// TIA Portal project "3 Animation final project" (V13)

(* hardware
DEVICE "S7-1200 station_1"  S7-1200 Station
   slot 0: "Rack_0"  Rack  V1.0
   slot 1: "PLC_1"  CPU 1212C AC/DC/Rly  6ES7 212-1BE40-0XB0  V4.1
DEVICE "HMI_1"  KTP400 Basic PN
   slot 0: "HMI"  HMI  6AV2 123-2DB03-0AX0  13.0.1.0
   slot 1: "HMI_RT_1"  KTP400 Basic PN  6AV2 123-2DB03-0AX0  13.0.1.0
   slot 5: "HMI_1.IE_CP_1"  PROFINET Interface
      slot 1: "PROFINET Interface_1"  PROFINET Interface
         slot 1: "Port_1"  Port
*)

// ===== PLC "PLC_1"  CPU 1212C AC/DC/Rly =====

VAR_GLOBAL   // PLC tag table "Default tag table"
   "Tag_1" AT %MD5 : DWord;
   "Tag_2" AT %MD0 : DWord;
   "Tag_4" AT %MW5 : Word;
   "Tag_3" AT %MW10 : Int;
   "Move box right" AT %M100.0 : Bool;
   "Motor up" AT %Q0.0 : Bool;
   "Move box left" AT %M100.1 : Bool;
   "Motor anti clockwise" AT %Q0.1 : Bool;
   "Tag_9" AT %MD5 : Time;
   "Tag_10" AT %MD12 : Real;
   "Tag_11" AT %MW15 : Int;
   "Capacitive Analog" AT %ID30 : DWord;
   "Tag_13" AT %MD22 : Real;
   "Capacitive Int" AT %MW50 : Word;
   "Motor clockwise" AT %Q0.2 : Bool;
   "Tank Level" AT %ID34 : DWord;
   "Tag_17" AT %MD25 : Real;
   "Tank Level scaled" AT %MD26 : Real;
   "Fill Valve" AT %QD30 : Real;
   "Drain Valve" AT %QD34 : Real;
   "Stop Filling Valve" AT %M200.0 : Bool;
   "Stop Draining Valve" AT %M200.1 : Bool;
   "Animation bit for filling" AT %M40.0 : Bool;
   "Clock_Byte" AT %MB300 : Byte;
   "Clock_10Hz" AT %M300.0 : Bool;
   "Clock_5Hz" AT %M300.1 : Bool;
   "Clock_2.5Hz" AT %M300.2 : Bool;
   "Clock_2Hz" AT %M300.3 : Bool;
   "Clock_1.25Hz" AT %M300.4 : Bool;
   "Clock_1Hz" AT %M300.5 : Bool;
   "Clock_0.625Hz" AT %M300.6 : Bool;
   "Clock_0.5Hz" AT %M300.7 : Bool;
   "Tag_21" AT %MB60 : Byte;
   "roller" AT %MD60 : Real;
   "roller_2" AT %MD70 : Real;
   "Tag_22" AT %MD65 : Real;
   "Tag_23" AT %MW60 : Int;
   "Tag_24" AT %MW65 : Int;
   "Down" AT %M90.0 : Bool;
   "Up" AT %M90.1 : Bool;
   "Door Animation Bit" AT %MW75 : Int;
   "Tag_26" AT %MW78 : Int;
   "Tag_27" AT %MW80 : Int;
   "Down(1)" AT %M90.2 : Bool;
   "Motor down" AT %Q0.3 : Bool;
   "Door Motor bit" AT %M101.0 : Bool;
END_VAR

// folder: System blocks/Program resources

DATA_BLOCK "IEC_Timer_0_DB"   // DB1
{ S7_Optimized_Access := 'FALSE' }
AUTHOR : Simatic
FAMILY : IEC
NAME : IEC_TMR
VERSION : 1.0
// stored: InstanceOfName ?
"?"
BEGIN
END_DATA_BLOCK

DATA_BLOCK "IEC_Timer_0_DB_1"   // DB2
{ S7_Optimized_Access := 'FALSE' }
AUTHOR : Simatic
FAMILY : IEC
NAME : IEC_TMR
VERSION : 1.0
// stored: InstanceOfName ?
"?"
BEGIN
END_DATA_BLOCK

DATA_BLOCK "IEC_Timer_0_DB_2"   // DB3
{ S7_Optimized_Access := 'FALSE' }
AUTHOR : Simatic
FAMILY : IEC
NAME : IEC_TMR
VERSION : 1.0
// stored: InstanceOfName ?
"?"
BEGIN
END_DATA_BLOCK

// folder: (top level)

FUNCTION "MHJ-PLC-Lab-Function-S71200" : Void   // FC1, SCL
{ S7_Optimized_Access := 'FALSE' }
VERSION : 0.1
BEGIN

   #Value := PEEK(area := 16#82,
                  dbNumber := 0,
                  byteOffset := 511);
   #Value := #Value + 1;

   POKE(area := 16#82,
        dbNumber := 0,
        byteOffset := 511,
        value := #Value);

   POKE(area := 16#81,
        dbNumber := 0,
        byteOffset := 1016,
        value := #Value_01_DW);
   POKE(area := 16#81,
        dbNumber := 0,
        byteOffset := 1020,
        value := #Value_02_DW);

   POKE(area := 16#81,
        dbNumber := 0,
        byteOffset := 511,
        value := B#16#00);

   FOR #forVal := 0 TO 120 DO
       FOR #forVal_2 := 0 TO 10 DO
           #rdTimeReturn := RD_SYS_T(#outputTime);
           #rdTimeReturn := WR_SYS_T(#outputTime);
           #rdTimeReturn := RD_SYS_T(#outputTime);
           #rdTimeReturn := WR_SYS_T(#outputTime);
       END_FOR;
       #SyncVal := PEEK(area := 16#81,
                        dbNumber := 0,
                        byteOffset := 511);
       IF #SyncVal = #CompVal THEN
           GOTO M_1;
       END_IF;
   END_FOR;
   RETURN;

   M_1:
   POKE(area := 16#81,
        dbNumber := 0,
        byteOffset := 511,
        value := B#16#0);
END_FUNCTION

ORGANIZATION_BLOCK "Main"   // OB1, LAD, ProgramCycle
TITLE = "Main Program Sweep (Cycle)"
{ S7_Optimized_Access := 'FALSE' }
VERSION : 0.1
   VAR_TEMP   // added for the SCL form of the ladder/FBD networks
      _w1 : Bool;
   END_VAR
BEGIN

REGION Network 1: Box Logic
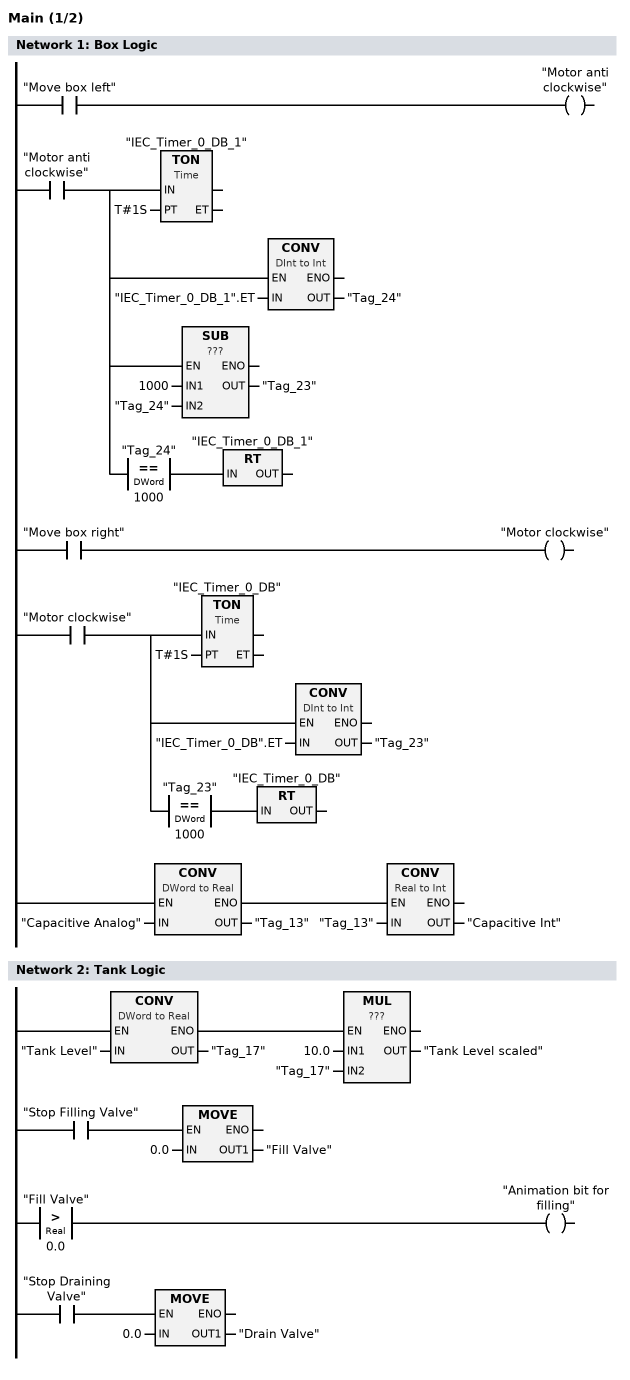
   // ENO of a box is taken as its EN; it also drops when the box reports an error
   "Motor anti clockwise" := "Move box left";
   "IEC_Timer_0_DB_1".TON(IN := "Motor anti clockwise", PT := T#1S);
   IF "Motor anti clockwise" THEN
       "Tag_24" := DINT_TO_INT("IEC_Timer_0_DB_1".ET);
       "Tag_23" := 1000 - "Tag_24";
   END_IF;
   IF "Motor anti clockwise" AND ("Tag_24" = 1000) THEN RESET_TIMER("IEC_Timer_0_DB_1"); END_IF;
   "Motor clockwise" := "Move box right";
   "IEC_Timer_0_DB".TON(IN := "Motor clockwise", PT := T#1S);
   IF "Motor clockwise" THEN "Tag_23" := DINT_TO_INT("IEC_Timer_0_DB".ET); END_IF;
   IF "Motor clockwise" AND ("Tag_23" = 1000) THEN RESET_TIMER("IEC_Timer_0_DB"); END_IF;
   "Tag_13" := DWORD_TO_REAL("Capacitive Analog");
   "Capacitive Int" := REAL_TO_INT("Tag_13");
END_REGION

REGION Network 2: Tank Logic
   RUNG wire#powerrail
      { S7_Templates := "[SrcType := DWord, DestType := Real]"; S7_GenerateENO := "TRUE" } Convert(in := "Tank Level", out => "Tag_17")
      { S7_Templates := "SrcType := ???"; S7_GenerateENO := "TRUE" } Mul(in1 := 10.0, in2 := "Tag_17", out => "Tank Level scaled")
   END_RUNG
   RUNG wire#powerrail
      Contact( "Stop Filling Valve" )
      { S7_GenerateENO := "TRUE" } Move(in := 0.0, out1 => "Fill Valve")
   END_RUNG
   RUNG wire#powerrail
      { S7_Templates := "SrcType := Real" } GT_Contact(in1 := "Fill Valve", in2 := 0.0)
      Coil( "Animation bit for filling" )
   END_RUNG
   RUNG wire#powerrail
      Contact( "Stop Draining Valve" )
      { S7_GenerateENO := "TRUE" } Move(in := 0.0, out1 => "Drain Valve")
   END_RUNG
   // the same network as SCL:
   // ENO of a box is taken as its EN; it also drops when the box reports an error
   "Tag_17" := DWORD_TO_REAL("Tank Level");
   "Tank Level scaled" := 10.0 * "Tag_17";
   IF "Stop Filling Valve" THEN "Fill Valve" := 0.0; END_IF;
   "Animation bit for filling" := "Fill Valve" > 0.0;
   IF "Stop Draining Valve" THEN "Drain Valve" := 0.0; END_IF;
END_REGION

REGION Network 3: Door Logic
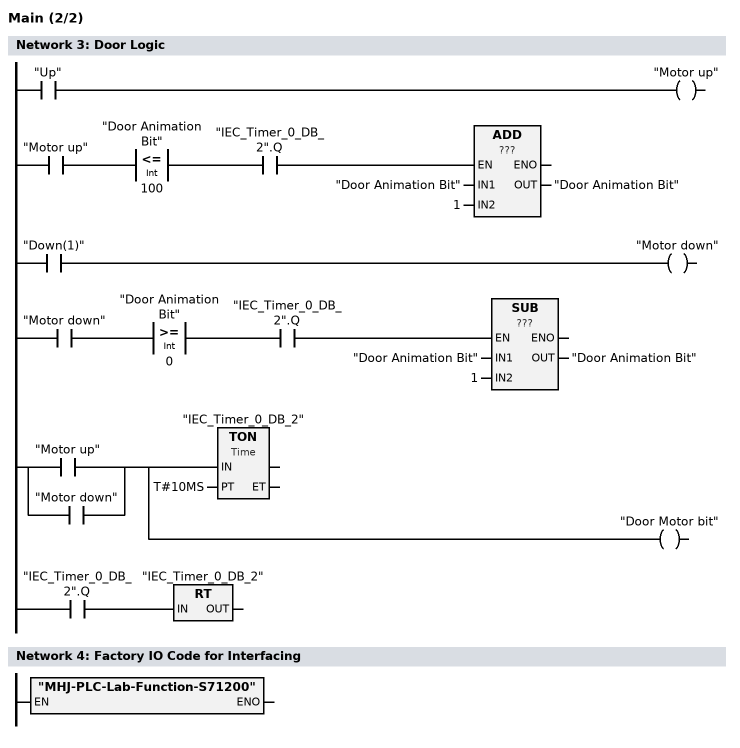
   "Motor up" := "Up";
   IF "Motor up" AND ("Door Animation Bit" <= 100) AND "IEC_Timer_0_DB_2".Q THEN
       "Door Animation Bit" := "Door Animation Bit" + 1;
   END_IF;
   "Motor down" := "Down(1)";
   IF "Motor down" AND ("Door Animation Bit" >= 0) AND "IEC_Timer_0_DB_2".Q THEN
       "Door Animation Bit" := "Door Animation Bit" - 1;
   END_IF;
   #_w1 := "Motor up" OR "Motor down";
   "IEC_Timer_0_DB_2".TON(IN := #_w1, PT := T#10MS);
   "Door Motor bit" := #_w1;
   IF "IEC_Timer_0_DB_2".Q THEN RESET_TIMER("IEC_Timer_0_DB_2"); END_IF;
END_REGION

REGION Network 4: Factory IO Code for Interfacing
   RUNG wire#powerrail
      "MHJ-PLC-Lab-Function-S71200"()
   END_RUNG
   // the same network as SCL:
   "MHJ-PLC-Lab-Function-S71200"();
END_REGION
END_ORGANIZATION_BLOCK

(* ===== HMI "HMI_RT_1" =====
connection "HMI_Connection_1": ETHERNET, SMART_S7_1200_OMS

HMI tags "Default tag table"
   "Tag_5" : Bool = PLC "Move box right", 100 ms
   "Tag_7" : Bool = PLC "Move box left", 100 ms
   "Tag_6" : Bool = PLC "Motor up", 100 ms
   "Tag_10" : Real = PLC "Tag_10", 100 ms
   "Tag_11" : Int = PLC "Tag_11", 100 ms
   "Tag_14" : Word = PLC "Capacitive Int", 100 ms
   "Tag_17" : Real = PLC "Tag_17", 100 ms
   "Tag_18" : Real = PLC "Tank Level scaled", 100 ms
   "Fill Valve" : Real = PLC "Fill Valve", 100 ms
   "Drain Valve" : Real = PLC "Drain Valve", 100 ms
   "Tag_19" : Bool = PLC "Stop Filling Valve", 100 ms
   "Tag_20" : Bool = PLC "Stop Draining Valve", 100 ms
   "Animation bit" : Bool = PLC "Animation bit for filling", 100 ms
   "Tag_13" : Real = PLC "Tag_13", 100 ms
   "Tag_21" : Byte = PLC "Tag_21", 100 ms
   "roller_HMI" : Real = PLC "roller", 100 ms
   "roller_2" : Real = PLC "roller_2", 100 ms
   "Tag_23" : Int = PLC "Tag_23", 100 ms
   "Tag_25" : Int = PLC "Door Animation Bit", 100 ms
   "Up" : Bool = PLC "Up", 100 ms
   "Down" : Bool = PLC "Down", 100 ms
   "Down(1)" : Bool = PLC "Down(1)", 100 ms
   "Door Motor bit" : Bool = PLC "Door Motor bit", 100 ms

graphic list "Valve": 0 'OFF'; 1..7 'Partially ON_1'; 8..10 'ON_1'

graphic list "Pipes": 0 'not flowing'; 1..7 'Partially flowing'; 8..10 'flowing'

graphic list "Roller": 0..249 '1'; 250..499 '2'; 500..749 '3'; 750..1000 '4'

graphic list "Motor": 0 'Graphic_24'; 1 'Graphic_25'

graphic list "Arrow": 0 'Graphic_27'; 1 'Graphic_26'

Template "Template_1" 480x272
   Button "Template_Button" at 388,227 size 63x44
   Button "Template_Button_3" at 28,227 size 63x44

screen "Root screen" 480x272, template "Template_1"
   Button "Button_5" at 202,139 size 122x32
   Button "Button_6" at 202,178 size 122x32
   TextField "Text field_1" at 149,97 size 224x32
   Button "Button_1" at 203,217 size 122x32
   GraphicView "Graphic view_1" at 223,8 size 83x67
   TextField "Text field_2" at 98,76 size 336x27

screen "Box" 480x272
   Button "Button_1" at 404,139 size 33x17
   Button "Button_2" at 33,139 size 33x19
   TextField "Text field_1" at 11,7 size 131x25
   Group "Group" at 33,133 size 404x46
   Button "Button_6" at 349,9 size 122x32
   Button "Button_3" at 404,236 size 67x32
   IOField "I/O field_1" at 66,109 size 39x32
   GraphicIOField "Graphic I/O field_1" at 35,170 size 32x28
   GraphicIOField "Graphic I/O field_2" at 409,170 size 32x28
   Button "Button_4" at 347,45 size 122x32

screen "Tank" 480x272
   Bar "Bar_1" at 254,70 size 120x139
   TextField "Text field_2" at 15,9 size 135x23
   GraphicView "Graphic view_1" at 254,54 size 122x18
   GraphicView "Graphic view_2" at 253,207 size 123x28
   Button "Button_4" at 429,184 size 45x23
   IOField "I/O field_1" at 383,54 size 43x29
   IOField "I/O field_2" at 383,181 size 43x29
   Button "Button_3" at 429,57 size 45x23
   IOField "I/O field_3" at 378,127 size 43x18
   GraphicView "Graphic view_5" at 295,28 size 33x28
   GraphicIOField "Graphic I/O field_1" at 387,21 size 39x32
   GraphicIOField "Graphic I/O field_2" at 385,224 size 39x32
   GraphicIOField "Graphic I/O field_3" at 327,35 size 62x13
   GraphicIOField "Graphic I/O field_4" at 424,35 size 56x13
   GraphicIOField "Graphic I/O field_5" at 325,239 size 62x13
   GraphicIOField "Graphic I/O field_6" at 422,239 size 58x13
   TextField "Text field_3" at 422,126 size 23x22
   GraphicView "Graphic view_3" at 303,233 size 23x25
   Button "Button_5" at 15,226 size 122x32
   Button "Button_1" at 15,148 size 67x32
   Button "Button_2" at 15,187 size 122x32

screen "Door" 480x272
   GraphicIOField "Graphic I/O field_1" at 10,106 size 63x27
   GraphicView "Graphic view_1" at 258,188 size 148x75
   GraphicView "Graphic view_2" at 206,106 size 44x46
   GraphicView "Graphic view_3" at 408,213 size 39x47
   Button "Button_1" at 206,158 size 41x43
   Button "Button_2" at 206,209 size 41x43
   Button "Button_3" at 406,7 size 67x32
   Button "Button_6" at 351,44 size 122x32
   Button "Button_5" at 351,84 size 122x32
   TextField "Text field_1" at 10,8 size 140x25
*)